FUNCTION_BLOCK EcSlaveDevFWUpdater EXTENDS FbBase
VAR CONSTANT	
	{attribute 'displaymode':='hexadecimal'} 
	COE_FWVERSION_OBJECT								: WORD := 16#100A;
END_VAR
VAR_OUTPUT CONSTANT
	MIN_SLAVE_DEV										:	INT := 1;
	MAX_SLAVE_DEV										:	INT := Param.ETHERCAT_SLAVE_DEV_FW_UPDATER_MAX_DEV;

	{attribute 'displaymode':='binary'}   
	MODE_READ											:	BYTE := 0;
	{attribute 'displaymode':='binary'}   
	MODE_WRITE											:	BYTE := 1;

	{attribute 'displaymode':='binary'}   
	OPTION_WRITE_FW_IF_VERSION_MATCH					:	BYTE := 2#0000_0001;
	
END_VAR
VAR_INPUT
{attribute 'displaymode':='binary'}         			
	Mode												:	BYTE  := 2#0000_0000; 

{attribute 'displaymode':='binary'}  	
	Options												:	BYTE  := 2#0000_0000; 		
				
	PathName											:	STRING; //Path incl. file name of FW file
	RegVersion											:	STRING; //Requested version
	ipSlaveInfoData										:	ARRAY [MIN_SLAVE_DEV..MAX_SLAVE_DEV] OF I_EcSlaveInfoData;
END_VAR
VAR_OUTPUT
	ActVersion											: ARRAY[MIN_SLAVE_DEV..MAX_SLAVE_DEV] OF STRING[20]; 	
	CntFWNOK											: INT; //Count of terminals FW not OK
	TermNo												: INT; //No of terminal in progress
	ProgressWriteFW										: UDINT;	
	VersionRead											: BOOL;
END_VAR
VAR
(*  Memory *****************************************************)
	lastState											: INT := 0;
	MinTerm												: INT;

(*  Timer ******************************************************)
(*  Trigger ****************************************************)

(*  Blocks *****************************************************)
	EcCoeSdoReadEx										: FB_EcCoeSdoReadEx := (nIndex := COE_FWVERSION_OBJECT, tTimeout := DEFAULT_ADS_TIMEOUT);

	CoEFwDownLoad										: FB_EcFoeLoad := (tTimeout := DEFAULT_ADS_TIMEOUT,dwPass := 0, eMode := eFoeMode_Write);
(*  Error ******************************************************)
(*  Dummys *****************************************************)
	{attribute 'hide' := ''}
	i,j													: INT := 0;

END_VAR

	(*********************************************************)
	
(* state machine ********************************************************)
	rtExecute(CLK := Execute);
	CASE state OF
	0 : 
		Busy 											:= FALSE;
		
		IF NOT Execute THEN
			Done 										:= FALSE;
			Error 										:= FALSE;
			ErrorID 									:= 0;
		END_IF
		IF rtExecute.Q THEN
			IF PathName = '' 
			THEN
				Error 									:= TRUE;
				ErrorID 								:= E_AdsErr.DEVICE_INVALIDPARM;

			ELSIF RegVersion = '' AND Mode = MODE_WRITE AND NOT Options.0
			THEN
 				Error 									:= TRUE;
				ErrorID 								:= E_AdsErr.DEVICE_INVALIDPARM; 
									
			ELSIF ipSlaveInfoData[MIN_SLAVE_DEV] = 0
			THEN
 				Error 									:= TRUE;
				ErrorID 								:= E_AdsErr.DEVICE_INVALIDPARM; 			
			ELSE
				Busy									:= TRUE;	
				Done 									:= FALSE;
				Error 									:= FALSE;
				ErrorID 								:= 0;
				TermNo									:= MIN_SLAVE_DEV;	
				ProgressWriteFW							:= 0;
				CntFWNOK								:= 0;					
				
			
				EcCoeSdoReadEx(bExecute := FALSE);
				CoEFwDownLoad(bExecute := FALSE);
				state									:= SEL(Mode = MODE_READ, 1, 2);
			END_IF
		END_IF
			
	1: (* Write FW *****************************************************************)
		CoEFwDownLoad(
			bExecute		:= ipSlaveInfoData[TermNo].rInfoData.AdsAddr.port <> 0 AND (ActVersion[TermNo] <> RegVersion OR Options.0) , 
			sNetId			:= F_CreateAmsNetId(nIds := ipSlaveInfoData[TermNo].rInfoData.AdsAddr.netId),
			nSlaveAddr		:= ipSlaveInfoData[TermNo].rInfoData.AdsAddr.port,
			sPathName		:= PathName,
			nProgress 		=> ProgressWriteFW);	
		IF NOT 	CoEFwDownLoad.bBusy
		THEN
			ProgressWriteFW								:= 0;
			IF CoEFwDownLoad.bError
			THEN
				ErrorID									:= EcCoESdoReadEx.nErrId;
				CntFWNOK								:= CntFWNOK + 1;	
				ActVersion[TermNo]						:= 'ERR_DOWNLOADING';
			ELSIF CoEFwDownLoad.bExecute	
			THEN
				ActVersion[TermNo]						:= 'DOWNLOADED';
			ELSE
				ActVersion[TermNo]						:= '------';
			END_IF
			//Next terminal
			TermNo										:= TermNo + 1;
			
			IF TermNo > MAX_SLAVE_DEV 
				OR ipSlaveInfoData[TermNo] = 0
			THEN //Start reading
				MEMSET(ADR(ActVersion),0,SIZEOF(ActVersion));
				VersionRead								:= FALSE;
				TermNo									:= MIN_SLAVE_DEV;		
				state									:= 2;
			END_IF		
			CoEFwDownLoad(bExecute := FALSE);
		ELSE
			ActVersion[TermNo]							:= CONCAT('DOWNLOADING ',CONCAT(TO_STRING(CoEFwDownLoad.nProgress),'%'));
		END_IF
	
	2: (* Read FW Version **********************************************************)
		EcCoESdoReadEx(
			bExecute		:= ipSlaveInfoData[TermNo].rInfoData.AdsAddr.port <> 0,
			sNetId			:= F_CreateAmsNetId(nIds := ipSlaveInfoData[TermNo].rInfoData.AdsAddr.netId),
			nSlaveAddr		:= ipSlaveInfoData[TermNo].rInfoData.AdsAddr.port,
			pDstBuf			:= ADR(ActVersion[TermNo]),
			cbBufLen		:= SIZEOF(ActVersion[TermNo]));
		IF NOT EcCoESdoReadEx.bBusy
		THEN
			IF EcCoESdoReadEx.bError 
			THEN
				ActVersion[TermNo]						:= 'ERR_READING';
				ErrorID									:= EcCoESdoReadEx.nErrId;
				CntFWNOK								:= CntFWNOK + 1;	
			ELSIF NOT EcCoESdoReadEx.bExecute 
			THEN
				ActVersion[TermNo]						:= 'NOT_CONNECTED';
			ELSIF ActVersion[TermNo] <> RegVersion
			THEN
				CntFWNOK								:= CntFWNOK + 1;	
			END_IF
			
			//Next terminal
			TermNo										:= TermNo + 1;
			
			IF TermNo > MAX_SLAVE_DEV
				OR ipSlaveInfoData[TermNo] = 0
			THEN
				TermNo									:= MAX_SLAVE_DEV;
				Done									:= CntFWNOK = 0;
				VersionRead								:= TRUE;
				Error									:= NOT Done;
				Busy									:= FALSE;
				state									:= 0;
			END_IF
			EcCoeSdoReadEx(bExecute := FALSE);
		END_IF
	END_CASE	

(* Record last state ******************************************)
IF state <> lastState AND state <> 0 AND NOT Error
THEN 
	lastState											:= state;
END_IF

(*************************************************************)

END_FUNCTION_BLOCK

(* stored: Version 1.1.0.1, ProductVersion 3.1.4024.5
   POU EcSlaveDevFWUpdater: Id {86a2a00d-90b4-44d2-b0de-15613e7ec3f5}, SpecialFunc None *)
